// TIA Portal V15.1 export
// export: Created 2020-06-12T07:35:54.8818359Z, ExportSetting None, DisplayName Totally Integrated Automation Portal, DisplayVersion V15.1, DisplayName TIA Portal Openness, DisplayVersion V15.1, DisplayName STEP 7 Professional, DisplayVersion V15.1, DisplayName STEP 7 Safety, DisplayVersion V15.1, DisplayName WinCC Advanced, DisplayVersion V15.1
FUNCTION "Desk_ES1GD02" : Void   // FC1211, FBD
TITLE = Control desk +ES1GD02 Lamp Control
{ S7_Optimized_Access := 'FALSE' }
// stored: AutoNumber false, SetENOAutomatically False
   VAR_TEMP
      _GD02_ltest : Bool;
      _GD02_elc_top : Bool;
      _GD02_elc_bot : Bool;
      _GD02_elc_lck : Bool;
   END_VAR
BEGIN

REGION Network 1: D06 LED Electrode carriage in Top position
   // "EQ_ESMLE1".M01.auto_on_R
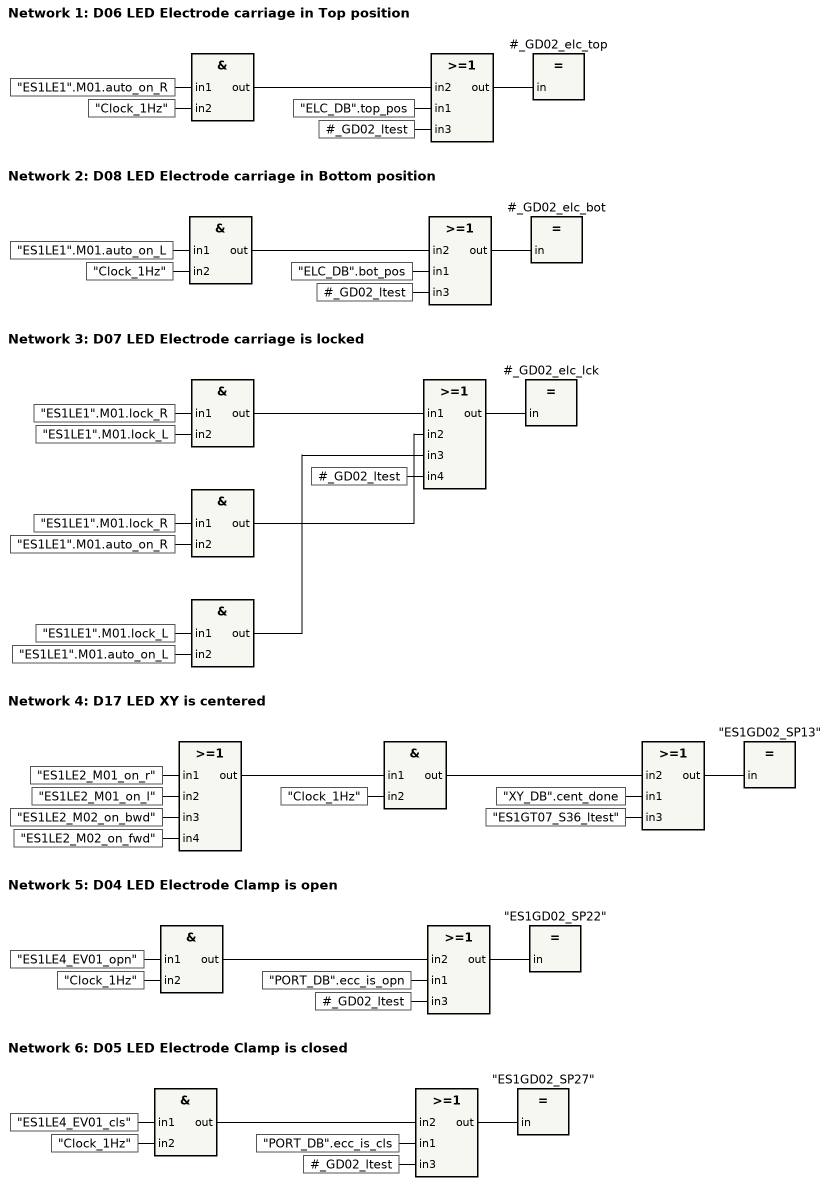
   #_GD02_elc_top := ("ES1LE1".M01.auto_on_R AND "Clock_1Hz") OR "ELC_DB".top_pos OR #_GD02_ltest;
END_REGION

REGION Network 2: D08 LED Electrode carriage in Bottom position
   // "ES1LE1".M01_run_left
   #_GD02_elc_bot := ("ES1LE1".M01.auto_on_L AND "Clock_1Hz") OR "ELC_DB".bot_pos OR #_GD02_ltest;
END_REGION

REGION Network 3: D07 LED Electrode carriage is locked
   // "ES1LE1".M01_run_right
   // "EQ_ESMLE1".M01.lock_L
   #_GD02_elc_lck := ("ES1LE1".M01.lock_R AND "ES1LE1".M01.lock_L) OR ("ES1LE1".M01.lock_R AND "ES1LE1".M01.auto_on_R) OR ("ES1LE1".M01.lock_L AND "ES1LE1".M01.auto_on_L) OR #_GD02_ltest;
END_REGION

REGION Network 4: D17 LED XY is centered
   "ES1GD02_SP13" := (("ES1LE2_M01_on_r" OR "ES1LE2_M01_on_l" OR "ES1LE2_M02_on_bwd" OR "ES1LE2_M02_on_fwd") AND "Clock_1Hz") OR "XY_DB".cent_done OR "ES1GT07_S36_ltest";
END_REGION

REGION Network 5: D04 LED Electrode Clamp is open
   "ES1GD02_SP22" := ("ES1LE4_EV01_opn" AND "Clock_1Hz") OR "PORT_DB".ecc_is_opn OR #_GD02_ltest;
END_REGION

REGION Network 6: D05 LED Electrode Clamp is closed
   "ES1GD02_SP27" := ("ES1LE4_EV01_cls" AND "Clock_1Hz") OR "PORT_DB".ecc_is_cls OR #_GD02_ltest;
END_REGION
END_FUNCTION
